KUKA KRL program: Thay_Mo.src, Thay_Mo.dat

--- Thay_Mo.src ---
&ACCESS RVP
&REL 1
&COMMENT Ve vi tri bom mo
DEF Thay_Mo()
  ;FOLD INI
    ;FOLD BASISTECH INI
      BAS(#INITMOV, 0)
    ;ENDFOLD
  ;ENDFOLD

  PTP HOME Vel=100% DEFAULT

  ; Di chuyen den vi tri bom mo
  PTP P_GREASE Vel=50% PDAT1 Tool[1] Base[0]

  ; Cho ky thuat vien thao tac
  HALT

  PTP HOME Vel=100% DEFAULT

END

--- Thay_Mo.dat ---
&ACCESS RV
&REL 1
DEFDAT Thay_Mo PUBLIC
  DECL E6POS HOME={A1 0.0, A2 -90.0, A3 90.0, A4 0.0, A5 0.0, A6 0.0}
  DECL E6POS P_GREASE={X 200.0, Y 0.0, Z 800.0, A 0.0, B 0.0, C 0.0, S 2, T 10}
ENDDAT
